(* CODESYS project proPlcPrg.export

Project tree, tasks and I/O mapping:
  program PLC_PRG [ST]
*)

// PLC_PRG
PROGRAM PLC_PRG
VAR
    iState   : INT := 0;
    rTargetX : REAL;
    rTargetY : REAL;
    rSpeed   : REAL := 1.0;
	i : INT;
	j : INT; 
	rPercent : REAL;
    byRed : BYTE;
    byGreen : BYTE;
	sCount : STRING;
    sMax : STRING;
	fbErrorTimer : TON;
END_VAR

// ---------------------------------------------------------
// 1. INITIALIZATION 
// ---------------------------------------------------------
IF GVL_Warehouse.arrWarehouse[1, 5].iMaxCapacity <> 5 THEN
    FOR i := 1 TO 5 DO
        FOR j := 1 TO 5 DO
             // Set Capacity: Col 1=1, Col 5=5
             GVL_Warehouse.arrWarehouse[i, j].iMaxCapacity := j; 
             
             // Reset everything else
             GVL_Warehouse.arrWarehouse[i, j].iCurrentCount := 0;
             GVL_Warehouse.arrWarehouse[i, j].dwColor := 16#FF00FF00; 
             GVL_Warehouse.arrWarehouse[i, j].sItemName := CONCAT('0 / ', INT_TO_STRING(j));
        END_FOR;
    END_FOR;
    iState := 0; // Ready to start
END_IF

// ---------------------------------------------------------
// 2. MAIN LOGIC
// ---------------------------------------------------------
CASE iState OF
    0: // IDLE (Handles both Auto and Manual inputs)
        // --- PATH A: AUTO ---
        IF GVL_Warehouse.xExecute THEN 
            GVL_Warehouse.xExecute := FALSE;
            GVL_Warehouse.iIncomingType := DWORD_TO_INT(TIME_TO_DWORD(TIME()) MOD 5) + 1;
            GVL_Warehouse.iTargetRow := GVL_Warehouse.iIncomingType;
            iState := 5; // Go to Search
        
        // --- PATH B: MANUAL ---
        ELSIF GVL_Warehouse.xManualExecute THEN 
            GVL_Warehouse.xManualExecute := FALSE;
            GVL_Warehouse.iIncomingType := GVL_Warehouse.iTargetRow; 
            iState := 6; // Go to Verify
        END_IF

        // Common Setup (Visuals)
        IF iState > 0 THEN
            CASE GVL_Warehouse.iIncomingType OF
                1: GVL_Warehouse.sIncomingName := 'Alpha';
                2: GVL_Warehouse.sIncomingName := 'Bravo';
                3: GVL_Warehouse.sIncomingName := 'Charlie';
                4: GVL_Warehouse.sIncomingName := 'Delta';
                5: GVL_Warehouse.sIncomingName := 'Echo';
                ELSE GVL_Warehouse.sIncomingName := 'Custom';
            END_CASE
            
            GVL_Warehouse.xBoxReady := TRUE;
            GVL_Warehouse.rActiveBoxX := GVL_Warehouse.rPickX;
            GVL_Warehouse.rActiveBoxY := GVL_Warehouse.rPickY;
            GVL_Warehouse.xCarrying := FALSE;
        END_IF

    5: // AUTO SEARCH (Find first empty column)
        GVL_Warehouse.iTargetCol := 0;
        FOR i := 1 TO 5 DO
            IF GVL_Warehouse.arrWarehouse[GVL_Warehouse.iTargetRow, i].iCurrentCount < GVL_Warehouse.arrWarehouse[GVL_Warehouse.iTargetRow, i].iMaxCapacity THEN
                GVL_Warehouse.iTargetCol := i;
                EXIT;
            END_IF;
        END_FOR;
        
        IF GVL_Warehouse.iTargetCol > 0 THEN iState := 10;
        ELSE GVL_Warehouse.xSystemFull := TRUE; iState := 0; END_IF

    6: // MANUAL VERIFY (Check if slot is valid)
        IF (GVL_Warehouse.iTargetRow < 1 OR GVL_Warehouse.iTargetRow > 5 OR GVL_Warehouse.iTargetCol < 1 OR GVL_Warehouse.iTargetCol > 5) OR
           (GVL_Warehouse.arrWarehouse[GVL_Warehouse.iTargetRow, GVL_Warehouse.iTargetCol].iCurrentCount >= GVL_Warehouse.arrWarehouse[GVL_Warehouse.iTargetRow, GVL_Warehouse.iTargetCol].iMaxCapacity) THEN
            GVL_Warehouse.xSystemFull := TRUE;
            iState := 0;
        ELSE
            iState := 10;
        END_IF

    10, 20, 40: // MOVEMENT ENGINE (Fast & Smooth)
        // 1. Set Targets
        IF iState = 10 THEN // To Dock
            GVL_Warehouse.rTargetX := GVL_Warehouse.rPickX;
            GVL_Warehouse.rTargetY := GVL_Warehouse.rPickY;
        ELSIF iState = 20 THEN // To Shelf
            GVL_Warehouse.rTargetX := (INT_TO_REAL(GVL_Warehouse.iTargetCol - 1) * 80.0) + 149.0;
            GVL_Warehouse.rTargetY := (INT_TO_REAL(GVL_Warehouse.iTargetRow - 1) * 60.0) + 135.0;
        ELSE // To Home
            GVL_Warehouse.rTargetX := GVL_Warehouse.rHomeX;
            GVL_Warehouse.rTargetY := GVL_Warehouse.rHomeY;
        END_IF

        // 2. Move (Proportional Speed)
        // This moves 20% of the remaining distance per cycle.
        GVL_Warehouse.rCraneX_Actual := GVL_Warehouse.rCraneX_Actual + (GVL_Warehouse.rTargetX - GVL_Warehouse.rCraneX_Actual) * 0.2;
        GVL_Warehouse.rCraneY_Actual := GVL_Warehouse.rCraneY_Actual + (GVL_Warehouse.rTargetY - GVL_Warehouse.rCraneY_Actual) * 0.2;

        // 3. Snap to Grid (Stop micro-decimals)
        IF ABS(GVL_Warehouse.rCraneX_Actual - GVL_Warehouse.rTargetX) < 1.0 THEN GVL_Warehouse.rCraneX_Actual := GVL_Warehouse.rTargetX; END_IF
        IF ABS(GVL_Warehouse.rCraneY_Actual - GVL_Warehouse.rTargetY) < 1.0 THEN GVL_Warehouse.rCraneY_Actual := GVL_Warehouse.rTargetY; END_IF

        // 4. Animation Sync
        IF iState = 20 THEN 
            GVL_Warehouse.rActiveBoxX := GVL_Warehouse.rCraneX_Actual;
            GVL_Warehouse.rActiveBoxY := GVL_Warehouse.rCraneY_Actual;
        END_IF

        // 5. Arrival Check
        IF GVL_Warehouse.rCraneX_Actual = GVL_Warehouse.rTargetX AND GVL_Warehouse.rCraneY_Actual = GVL_Warehouse.rTargetY THEN
            IF iState = 10 THEN
                GVL_Warehouse.xCarrying := TRUE;
                GVL_Warehouse.xBoxReady := FALSE;
                iState := 20;
            ELSIF iState = 20 THEN iState := 30;
            ELSE iState := 0; END_IF
        END_IF

    30: // UPDATE DATA
        // Increment Count
        GVL_Warehouse.arrWarehouse[GVL_Warehouse.iTargetRow, GVL_Warehouse.iTargetCol].iCurrentCount := GVL_Warehouse.arrWarehouse[GVL_Warehouse.iTargetRow, GVL_Warehouse.iTargetCol].iCurrentCount + 1;
        
        // Update Text
        GVL_Warehouse.arrWarehouse[GVL_Warehouse.iTargetRow, GVL_Warehouse.iTargetCol].sItemName := 
        CONCAT(CONCAT(INT_TO_STRING(GVL_Warehouse.arrWarehouse[GVL_Warehouse.iTargetRow, GVL_Warehouse.iTargetCol].iCurrentCount), ' / '), INT_TO_STRING(GVL_Warehouse.arrWarehouse[GVL_Warehouse.iTargetRow, GVL_Warehouse.iTargetCol].iMaxCapacity));
        
        // Update Color
        IF GVL_Warehouse.arrWarehouse[GVL_Warehouse.iTargetRow, GVL_Warehouse.iTargetCol].iMaxCapacity > 0 THEN
            rPercent := INT_TO_REAL(GVL_Warehouse.arrWarehouse[GVL_Warehouse.iTargetRow, GVL_Warehouse.iTargetCol].iCurrentCount) / INT_TO_REAL(GVL_Warehouse.arrWarehouse[GVL_Warehouse.iTargetRow, GVL_Warehouse.iTargetCol].iMaxCapacity);
        ELSE rPercent := 1.0; END_IF
        
        GVL_Warehouse.arrWarehouse[GVL_Warehouse.iTargetRow, GVL_Warehouse.iTargetCol].dwColor := SHL(DWORD#16#FF, 24) OR SHL(REAL_TO_DWORD(255.0 * rPercent), 16) OR SHL(REAL_TO_DWORD(255.0 * (1.0 - rPercent)), 8);
        
        GVL_Warehouse.xCarrying := FALSE;
        iState := 40;
END_CASE
fbErrorTimer(IN := GVL_Warehouse.xSystemFull, PT := T#2S);

// 2. If the timer finishes (2 seconds passed), turn off cell full warning
IF fbErrorTimer.Q THEN
    GVL_Warehouse.xSystemFull := FALSE;
END_IF

END_PROGRAM
